INTERFACE IF_FillRegister EXTENDS __SYSTEM.IQueryInterface

METHOD put : BOOL
VAR_INPUT
	i_diInValue : DINT;
END_VAR
END_METHOD

PROPERTY xReadyForPut : BOOL
GET
END_GET
END_PROPERTY

END_INTERFACE

(* stored: Version 1.1.0.1
   Itf IF_FillRegister: Id {299b3917-73bb-40dd-bcb2-27c95399145d}
   Method put: Id {f9aa1693-d4c1-42e9-a1d9-c01823c4d16b}
   Property xReadyForPut: Id {c56654b4-25a2-44f8-a355-c51ded9360cc}
   Get Get: Id {962aaede-243d-467f-b0be-c4a817184d53} *)
